Universal Robots PolyScope program: a.urp

Program a (installation=default directory=/programs createdIn=5.2.0.61336 lastSavedIn=5.2.0.61336 robotSerialNumber=20195500451)
Calibrated DH parameters: a=[0.00002, -0.231658, -0.317125, 0.000011, 0.000055, 0]; d=[0.162082, 123.190176, -180.284242, 57.22734, 0.099524, 0.09934]; alpha=[1.569304, 0.00289, 0.004025, 1.569925, -1.569026, 0]; deltaTheta=[0, 0.993923, 4.662183, 0.627072, 0.000001, 0]
Robot Program (runOnlyOnce=false)
  MoveJ speed 60 deg/s, acceleration 80 deg/s^2 (useActiveTCP=true positionType=JointAngles) feature=Base
    Waypoint Waypoint_1: TCP in base x=366.156 y=-232.145 z=399.282 mm, rx=1.3632 ry=-0.93 rz=0.935 rad; joints [0, -77.43, -123.769, -90.009, 0.001, -0.002] deg
